(* Logix 5000 project; controller ExampleFile_V32 vendor 1 type 14 code 222 rev 32.11; software revision 32.00 *)

TASK MainTask (continuous, watchdog 500 ms) : MainProgram
TASK SafetyTask (periodic, rate 20 ms, priority 10, watchdog 20 ms, safety) : SafetyProgram

MODULES
   Local : vendor 1 type 14 code 222 (5069 0, rev 32.11)
END_MODULES

TYPE CommandString :   // Premixer command string based on CommandString.xlsx
STRUCT
   Cmd : STRING[10];
   Value : DINT[10];
END_STRUCT
END_TYPE

TYPE ISA88_PackML_Cmd :
STRUCT
   ClearFaults : BOOL;   // Program call to ClearFaults
   Clearing_ons : BOOL;   // Initialize to ClearFaults
   Hold_EM_Clear : TIMER;   // Holding time EM_Clear
   Resetting : BOOL;   // Program call to Resetting
   Resetting_ons : BOOL;   // Initialize Resetting
   Starting : BOOL;   // Program call to Starting
   Starting_ons : BOOL;   // Initialize Starting
   Stopping : BOOL;   // Program call to Stopping
   Stopping_ons : BOOL;   // Initialize Stopping
END_STRUCT
END_TYPE

TYPE ISA88_PackML_PackTags_Command :
STRUCT
   OpperationMode : ISA88_PackML_PackTags_Command_Opperation;   // Forces mode to obj model
   StateTransmittion : ISA88_State_UserInputs;
   Recept : DINT;   // currently not in use
END_STRUCT
END_TYPE

TYPE ISA88_PackML_PackTags_Command_Opperation :
STRUCT
   Automatic : BOOL;   // Forces mode to Automatic
   Maintenance : BOOL;   // Forces mode to Maintenance
   Manual : BOOL;   // Forces mode to Manual
   Cleaning : BOOL;   // Forces mode to Cleaning
   MES_Controlled : BOOL;   // Forces mode to CustomerDefined1
   CustomerDefined2 : BOOL;   // Forces mode to CustomerDefined2
END_STRUCT
END_TYPE

TYPE ISA88_PackML_PackTags_Status_Mode :   // Feedback which mode is active
STRUCT
   Automatic : BOOL;   // Current mode is Automatic
   Maintenance : BOOL;   // Current mode is Maintenance
   Manual : BOOL;   // Current mode is Manual
   Cleaning : BOOL;   // Current mode is Cleaning
   MES_Controlled : BOOL;   // Current mode is CustomerDefined1
   CustomerDefined2 : BOOL;   // Current mode is CustomerDefined2
END_STRUCT
END_TYPE

TYPE ISA88_PackML_SEQ :
STRUCT
   Clear : DINT;   // Clearing step number
   Resetting : DINT;   // Resetting step number
   Starting : DINT;   // Starting step number
   Stopping : DINT;   // Stopping step number
END_STRUCT
END_TYPE

TYPE ISA88_PackML_STS :
STRUCT
   ClearSeq_PC : BOOL;   // Clearing complete
   CompletingSeq_PC : BOOL;   // Completing complete
   ResettingSeq_PC : BOOL;   // Resetting complete
   StartingSeq_PC : BOOL;   // Starting complete
   StoppingSeq_PC : BOOL;   // Stopping complete
END_STRUCT
END_TYPE

TYPE ISA88_State_SC :
STRUCT
   Execute_to_Completing : BOOL;   // EquipmentModule requests to move from Execute to Completing
   Unholding_to_Execute : BOOL;   // EquipmentModule requests to move from Unholding to Execute
   Starting_to_Execute : BOOL;   // EquipmentModule requests to move from Starting to Execute
   Holding_to_Held : BOOL;   // EquipmentModule requests to move from Holding to Held
   Completing_to_Completed : BOOL;   // EquipmentModule requests to move from Completing to Completed
   Suspending_to_Suspended : BOOL;   // EquipmentModule requests to move from Suspending to Suspended
   Unsuspending_to_Execute : BOOL;   // EquipmentModule requests to move from Unsuspending to Execute
   Resetting_to_Idle : BOOL;   // EquipmentModule requests to move from Resetting to Idle
   Stopping_to_Stopped : BOOL;   // EquipmentModule requests to move from Stopping to Stopped
   Clearing_to_Stopped : BOOL;   // EquipmentModule requests to move from Clearing to Stopped
   Aborting_to_Aborted : BOOL;   // EquipmentModule requests to move from Aborting to Aborted
   Wrk_Module_Disabled : BOOL;   // Disables the module
   Wrk_Stop_trigger : BOOL;   // Forces the module to Stopped
   Wrk_Abort_trigger : BOOL;   // Forces the module to fault
   Sts_CurrentJob : STRING;   // Description of current job
   Wrk_Suspend : BOOL;   // Forces the module to suspend
   Wrk_Unsuspend : BOOL;   // Forces the module to Execute from Suspend
END_STRUCT
END_TYPE

TYPE ISA88_State_UserInputs :   // operations from the HMI
STRUCT
   Hold : BOOL;
   UnHold : BOOL;
   Start : BOOL;
   Suspend : BOOL;
   UnSuspend : BOOL;
   Reset : BOOL;
   Stop : BOOL;
   Abort : BOOL;
   Clear : BOOL;
END_STRUCT
END_TYPE

TYPE ISA88_State_UserOutputs :
STRUCT
   Held : BOOL;
   Unholding : BOOL;
   Holding : BOOL;
   Idle : BOOL;
   Starting : BOOL;
   Execute : BOOL;
   Completing : BOOL;
   Complete : BOOL;
   Resetting : BOOL;
   Unsuspending : BOOL;
   Suspended : BOOL;
   Suspending : BOOL;
   Stopped : BOOL;
   Stopping : BOOL;
   Clearing : BOOL;
   Aborted : BOOL;
   Aborting : BOOL;
END_STRUCT
END_TYPE

TYPE STRING16 :
STRUCT
   LEN : DINT;
   DATA : SINT[16];
END_STRUCT
END_TYPE

ADD_ON_INSTRUCTION ClearString   (* revision 1.0 *)
VAR_INPUT
   StartValue : DINT; {visible}
   final_value : DINT; {visible}
END_VAR
VAR_IN_OUT
   String : STRING[100]; {required}
END_VAR
VAR_INPUT
   cmd_Clear : BOOL; {visible}
END_VAR
VAR
   i : DINT; {access None}   // local index
END_VAR

ROUTINE Logic   (* structured text *)
   ////////////////////////////////////////////////////////////
   //   Copyright (c)
   //------------------------------------------------------------
   //   Routine: ClearString - Logic
   //   Author: WPI\tom.reit
   //   Created: 19-5-2022
   //------------------------------------------------------------
   //   Description:
   //
   //
   //   History:
   //
   ////////////////////////////////////////////////////////////
   if cmd_Clear then
   	for i := StartValue to final_value do
   		String[i]:='';
   	end_for;
   	cmd_Clear:=0;
   end_if;
END_ROUTINE
END_ADD_ON_INSTRUCTION

ADD_ON_INSTRUCTION Command_String   (* revision 1.0, vendor WPI, ExecutePrescan *)
// Mixer control based on Orklas command string.
// Revision note:
// First version
VAR_IN_OUT
   CommandString : STRING; {required}   // Input Command string
END_VAR
VAR_OUTPUT
   Cmd_Mixer : INT; {visible}   // bit 0 = stop mixer bit 1 = start mixer bit 2 = open mixer bit 3 = close mixer bit 4 = manual step bit 5 = discharge
   Cmd_Mixer_Speed_Fast : DINT; {visible}
   Cmd_Mixer_Time_Fast : DINT; {visible}
   Cmd_Mixer_Time_Slow : DINT; {visible}
   Cmd_Mixer_Time_Wait : DINT; {visible}
   Cmd_Mixer_Temperature : REAL; {visible}
   Cmd_Mixer_Time_Min : DINT; {visible}   // minimal mixing time
   Cmd_Mixer_Time_Max : DINT;   // max mixing time
   Sts_Time_RecievedCommand : LINT; {visible}
   Sts_Time_WriteCommand : LINT; {visible}
   Sts_MixingByTime : BOOL; {visible}
   Sts_MixingByTemperature : BOOL; {visible}
   Sts_SuccesfulRead : BOOL; {visible}   // String was succesful read and write according to CommandString
   ERR_InvalidCommand : BOOL; {visible}   // command didnt have end token
   ERR_TooManySegments : BOOL; {visible}   // Segment index reached higher than max value
   Cmd_Mixer_Speed_Slow : DINT; {visible}
END_VAR
VAR
   CommandString_Segment : STRING[10] := ([0] := 'MBD', [1] := 'MC', [2] := 'MSF', [3] := 'MTF');
   CommandString_Segment_Value : STRING[10] := ([0] := '1', [1] := '1', [2] := '80', [3] := '100');
   CommandStringSize : DINT := 26;
   count : INT := 82;
   i : INT;
   FoundPlace : DINT := 4;
   prev_i : DINT := 26;
   readString : BOOL;
   segment_Index : INT := 4;   // index num for array
   wrk_end_token : SINT := '#';   // end token will always be " # "
   wrk_split_token : SINT := ';';
   sts_CommandString : CommandString := (Cmd[0] := 'MBD', Cmd[1] := 'MC', Cmd[2] := 'MSF', Cmd[3] := 'MTF', Value[0] := 1, Value[1] := 1, Value[2] := 80, Value[3] := 100);
   wrk_String : STRING;   // temp string will be overwritten by each segment
   wrk_value_token_str : STRING := '_';
   wrk_Prev_CommandString : STRING;
END_VAR

ROUTINE Logic   (* structured text *)
// Mixer control based on Orklas command string.
   ////////////////////////////////////////////////////////////
   //   Copyright (c)  WPI
   //------------------------------------------------------------
   //   Routine: Command_String - Logic
   //   Author: WPI\engineer
   //   Created: 29-9-2021
   //------------------------------------------------------------
   //   Description:
   //           Mixer control based on Orklas command string.
   //
   //
   //   History:
   //
   ////////////////////////////////////////////////////////////
   #region "Check for new command"
   	if wrk_Prev_CommandString <> CommandString then
   		Sts_SuccesfulRead	:=0;
   		readString			:=1;
   		gsv(WallClockTime,,CurrentValue,Sts_Time_RecievedCommand);
   	end_if;
   #endregion
   #region "Read command string and apply logic"
   	if readString then
   	#region "Check if command is valid"
   		for i := 0 to 81 do
   			if CommandString.DATA[i] = wrk_end_token then
   				CommandStringSize		:=	i;	// set comamndstringSize
   				ERR_InvalidCommand		:=	0;	// valid string detected
   				exit;							// break for loop
   			end_if;
   			if i=81 AND CommandString.DATA[i] <> wrk_end_token then
   				ERR_InvalidCommand		:=	1; 	// no # was found in command string
   				readString				:=	0;	// break readstring
   			end_if;
   		end_for;
   				i						:=	0;	// set index back to 0
   	#endregion
   	#region Clear old Segments
   		for i := 0 to 9 do
   			Cmd_Mixer										:=0;
   			Cmd_Mixer_Speed_Fast							:=0;
   			Cmd_Mixer_Speed_Slow							:=0;
   			Cmd_Mixer_Temperature							:=0;
   			Cmd_Mixer_Time_Fast								:=0;
   			Cmd_Mixer_Time_Max								:=0;
   			Cmd_Mixer_Time_Min								:=0;
   			Cmd_Mixer_Time_Slow								:=0;
   			Cmd_Mixer_Time_Wait								:=0;
   			CommandString_Segment[i]						:='';
   			sts_CommandString.Cmd[i]						:='';
   			for count := 0 to 81 do
   				CommandString_Segment[i].DATA[count]		:=0;
   				sts_CommandString.Cmd[i].DATA[count]		:=0;
   				CommandString_Segment[i].LEN				:=0;
   				sts_CommandString.Cmd[i].LEN				:=0;
   				CommandString_Segment_Value[i].DATA[count]	:=0;
   				sts_CommandString.Cmd[i].DATA[count]		:=0;
   				CommandString_Segment_Value[i].LEN 			:=0;
   				sts_CommandString.Cmd[i].LEN 				:=0;
   			end_for;
   		end_for;
   		i:=0;
   	#endregion
   	#region ReadString
   		prev_i			:=	0;	// prepre for new string
   		segment_Index	:=	0;	// prepare for new string
   		for i := 0 to CommandStringSize do
   			wrk_String.DATA[i-prev_i]	:=	CommandString.DATA[i];
   			wrk_String.LEN				:=	i-prev_i;
   			if CommandString.DATA[i] = wrk_split_token  then
   				prev_i:=(i+1);
   				#region Prevent overflow array
   					if segment_Index>9 then
   						ERR_TooManySegments	:=1;
   						readString			:=0;
   						exit;
   					else
   						ERR_TooManySegments:=0;
   					end_if;
   				#endregion
   				CommandString_Segment[segment_Index]:=wrk_String;
   				segment_Index:=segment_Index+1;
   			end_if;
   		end_for;
   	#endregion
   	if NOT ERR_TooManySegments AND NOT ERR_InvalidCommand THEN
   		/* Clear wrk_string*/
   		wrk_String		:=	'';
   		wrk_String.LEN	:=	0;
   		#region read cmd value
   		FoundPlace:=0;
   		i:=0;
   			for i := 0 to segment_Index-1 do
   				find(CommandString_Segment[i],wrk_value_token_str,1,FoundPlace);
   				for count := FoundPlace to CommandString_Segment[i].LEN do
   					CommandString_Segment_Value[i].DATA[count-FoundPlace]:=CommandString_Segment[i].DATA[count];
   					CommandString_Segment_Value[i].LEN:=CommandString_Segment[i].LEN-FoundPlace;
   				end_for;
   			end_for;
   			i		:=	0;
   			count	:=	0;
   		#endregion
   		#region SubString
   			for i := 0 to segment_Index-1 do
   				find(CommandString_Segment[i],wrk_value_token_str,1,FoundPlace);
   				for count := FoundPlace-1 to 81 do
   					CommandString_Segment[i].DATA[count]:=0;
   				end_for;
   				CommandString_Segment[i].LEN:=FoundPlace-1;
   			end_for;
   		#endregion
   		#region Move values to sturcture
   			for i := 0 to segment_Index-1 do
   				sts_CommandString.Cmd[i]	:=	CommandString_Segment[i];
   				STOD(CommandString_Segment_Value[i],sts_CommandString.Value[i]);
   			end_for;
   		#endregion
   		#region "decode string"
   			for i := 0 to 9 do
   				if 		sts_CommandString.Cmd[i] 		= 	'MBD' 	then 	// Mixing by time / duration
   							Sts_MixingByTime:=1;
   							Sts_MixingByTemperature:=0;
   				elsif 	sts_CommandString.Cmd[i] 		= 	'MBT' 	then 	// Mixing by temperature
   							Sts_MixingByTime:=0;
   							Sts_MixingByTemperature:=1;
   				elsif 	sts_CommandString.Cmd[i] 		= 	'MC' 	then 	// Mixing Command
   					if		sts_CommandString.Value[i]	= 	0 		then	// Stop Mixer
   						Cmd_Mixer:=2#0000_0000_0000_0001;
   					elsif	sts_CommandString.Value[i]	= 	1 		then	// Start Mixer
   						Cmd_Mixer:=2#0000_0000_0000_0010;
   					elsif	sts_CommandString.Value[i]	= 	2 		then	// open Mixer
   						Cmd_Mixer:=2#0000_0000_0000_0100;
   					elsif	sts_CommandString.Value[i]	= 	3 		then	// close Mixer
   						Cmd_Mixer:=2#0000_0000_0000_1000;
   					elsif	sts_CommandString.Value[i]	= 	4 		then	// manual step active
   						Cmd_Mixer:=2#0000_0000_0001_0000;
   					elsif	sts_CommandString.Value[i]	= 	5 		then	// discharge mixer
   						Cmd_Mixer:=2#0000_0000_0010_0000;
   					end_if;
   				elsif 	sts_CommandString.Cmd[i] 		= 	'MSF' 	then 	// Mixer speed fast
   							Cmd_Mixer_Speed_Fast:=sts_CommandString.Value[i];
   				elsif 	sts_CommandString.Cmd[i] 		= 	'MSS' 	then 	// Mixer speed slow
   							Cmd_Mixer_Speed_Slow:=sts_CommandString.Value[i];
   				elsif 	sts_CommandString.Cmd[i] 		= 	'MTF' 	then 	// Mixing time fast
   							Cmd_Mixer_Time_Fast:=sts_CommandString.Value[i];
   				elsif 	sts_CommandString.Cmd[i] 		= 	'MTS' 	then 	// Mixing time slow
   							Cmd_Mixer_Time_Slow:=sts_CommandString.Value[i];
   				elsif 	sts_CommandString.Cmd[i] 		= 	'MTW' 	then 	// Waiting time
   							Cmd_Mixer_Time_Wait:=sts_CommandString.Value[i];
   				elsif 	sts_CommandString.Cmd[i] 		= 	'MOT' 	then 	// Optimal mixing temperature
   							Cmd_Mixer_Temperature:=sts_CommandString.Value[i];
   				elsif 	sts_CommandString.Cmd[i] 		= 	'MIT' 	then 	// Min mixing time
   							Cmd_Mixer_Time_Min:=sts_CommandString.Value[i];
   				elsif 	sts_CommandString.Cmd[i] 		= 	'MAT' 	then 	// Max mixing time
   							Cmd_Mixer_Time_Max:=sts_CommandString.Value[i];
   				end_if;
   			end_for;
   			Sts_SuccesfulRead:=1;
   			gsv(WallClockTime,,CurrentValue,Sts_Time_WriteCommand);
   		end_if;
   	#endregion
   	i:=0;
   	readString:=0;
   	wrk_Prev_CommandString:=CommandString;
   	end_if;
   #endregion
   
END_ROUTINE

ROUTINE Prescan   (* structured text *)
   ////////////////////////////////////////////////////////////
   //   Copyright (c)  WPI
   //------------------------------------------------------------
   //   Routine: Prescan
   //   Author: WPI\engineer
   //   Created: 29-9-2021
   //------------------------------------------------------------
   //   Description:
   //
   //
   //   History:
   //
   ////////////////////////////////////////////////////////////
   wrk_end_token		:=35; // 35 is # ascii
   wrk_split_token		:=59; // 35 is # ascii
   wrk_value_token_str	:='_';// _ is value token
   
   
END_ROUTINE
END_ADD_ON_INSTRUCTION

ADD_ON_INSTRUCTION CountUpAndDown   (* revision 1.0, vendor WPI *)
VAR_INPUT
   CountingSpeed : DINT; {visible}   // in miliseconds
END_VAR
VAR_OUTPUT
   Count : DINT; {visible}
END_VAR
VAR_INPUT
   MaxCount : DINT := 10; {visible}   // max value to count to
   Holding_Time : DINT := 2500; {visible}   // in milisec
END_VAR
VAR_OUTPUT
   Done : BOOL; {visible}
END_VAR
VAR
   Time_puls : TIMER := (PRE := 500); {access None}
   count_UP : BOOL := 1; {access None}
   holdingtime : TIMER[2]; {access None}
END_VAR

ROUTINE Logic   (* ladder *)
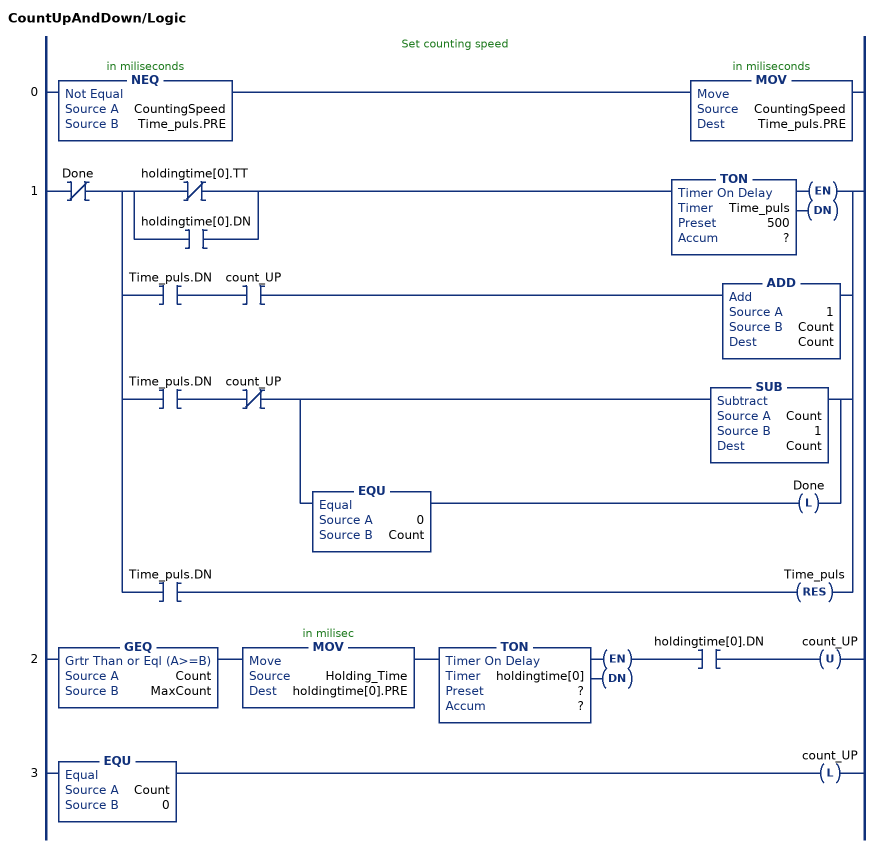
   // Set counting speed
   0: NEQ(CountingSpeed,Time_puls.PRE)MOV(CountingSpeed,Time_puls.PRE);
   1: XIO(Done)[[XIO(holdingtime[0].TT) ,XIC(holdingtime[0].DN) ] TON(Time_puls,?,?) ,XIC(Time_puls.DN) XIC(count_UP) ADD(1,Count,Count) ,XIC(Time_puls.DN) XIO(count_UP) [SUB(Count,1,Count) ,EQU(0,Count) OTL(Done) ] ,XIC(Time_puls.DN) RES(Time_puls) ];
   2: GEQ(Count,MaxCount)MOV(Holding_Time,holdingtime[0].PRE)TON(holdingtime[0],?,?)XIC(holdingtime[0].DN)OTU(count_UP);
   3: EQU(Count,0)OTL(count_UP);
END_ROUTINE
END_ADD_ON_INSTRUCTION

ADD_ON_INSTRUCTION CREATE_MERKER   (* revision 1.0 *)
VAR_INPUT
   INPUT : BOOL := 1; {required}
   RESET : BOOL; {required}
END_VAR
VAR_OUTPUT
   MERKER : BOOL; {access Read Only, visible}
END_VAR
VAR_INPUT
   I_NORMALY_OPEN : BOOL; {required}
END_VAR

ROUTINE Logic   (* ladder *)
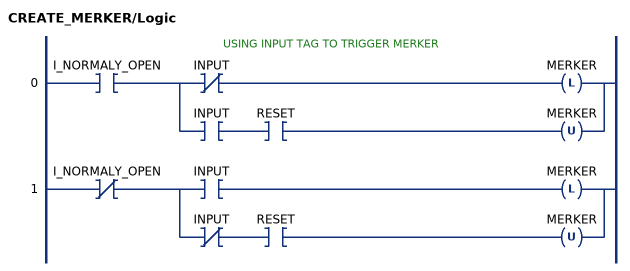
   // USING INPUT TAG TO TRIGGER MERKER
   0: XIC(I_NORMALY_OPEN)[XIO(INPUT) OTL(MERKER) ,XIC(INPUT) XIC(RESET) OTU(MERKER) ];
   1: XIO(I_NORMALY_OPEN)[XIC(INPUT) OTL(MERKER) ,XIO(INPUT) XIC(RESET) OTU(MERKER) ];
END_ROUTINE
END_ADD_ON_INSTRUCTION

ADD_ON_INSTRUCTION Dryrun_Sensor   (* revision 1.0, vendor WPI, ExecutePrescan *)
// Help:
// Geeft een alarm als de dryrun sensor 0 is en de pomp stuur waarde1 is.
VAR_INPUT
   I_DryrunSensor : BOOL; {required}
   I_PumpRunning : BOOL; {required}
END_VAR
VAR_OUTPUT
   Alarm : BOOL; {visible}   // Dryun is active
END_VAR
VAR_INPUT
   Reset : BOOL; {required}   // Reset the alarm if active
END_VAR
VAR
   DryrunTimer : TIMER := (PRE := 5000); {access None}
   ons : DINT; {access None}
END_VAR

ROUTINE Logic   (* ladder *)
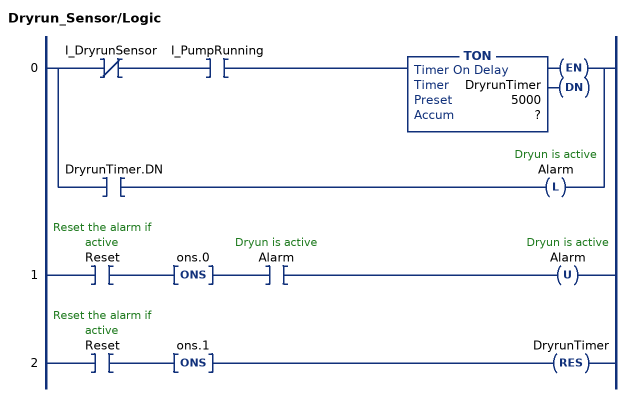
   0: [XIO(I_DryrunSensor) XIC(I_PumpRunning) TON(DryrunTimer,?,?) ,XIC(DryrunTimer.DN) OTL(Alarm) ];
   1: XIC(Reset)ONS(ons.0)XIC(Alarm)OTU(Alarm);
   2: XIC(Reset)ONS(ons.1)RES(DryrunTimer);
END_ROUTINE

ROUTINE Prescan   (* structured text *)
// sets timer
   DryrunTimer.PRE :=5000;		// set dryrun timer to 5 sec
END_ROUTINE
END_ADD_ON_INSTRUCTION

ADD_ON_INSTRUCTION FLIP_FLOP   (* revision 1.0 *)
VAR_INPUT
   input_time : DINT := 1500;
END_VAR
VAR_OUTPUT
   Q : BOOL; {access Read Only, visible}
   QB : BOOL; {access Read Only, visible}
END_VAR
VAR_INPUT
   INPUT_TIME_Q : DINT; {required}   // the time Q is going to be active
   INPUT_TIME_QB : DINT; {required}   // the time QB is going to be active
END_VAR
VAR
   FLIPFLOP_TIME : DINT; {access None}
   FLIPFLOP_timer1 : TIMER; {access None}
   FLIPFLOP_timer2 : TIMER := (PRE := 7500); {access None}
   FLIPFLOP_TIME1 : DINT; {access None}
   FLIPFLOP_TIME2 : DINT; {access None}
END_VAR

ROUTINE Logic   (* ladder *)
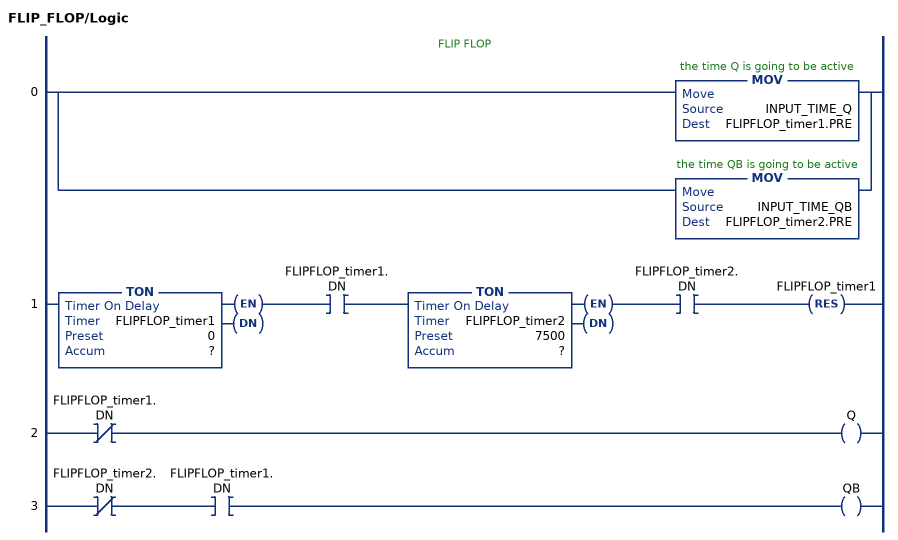
   // FLIP FLOP
   0: [MOV(INPUT_TIME_Q,FLIPFLOP_timer1.PRE) ,MOV(INPUT_TIME_QB,FLIPFLOP_timer2.PRE) ];
   1: TON(FLIPFLOP_timer1,?,?)XIC(FLIPFLOP_timer1.DN)TON(FLIPFLOP_timer2,?,?)XIC(FLIPFLOP_timer2.DN)RES(FLIPFLOP_timer1);
   2: XIO(FLIPFLOP_timer1.DN)OTE(Q);
   3: XIO(FLIPFLOP_timer2.DN)XIC(FLIPFLOP_timer1.DN)OTE(QB);
END_ROUTINE
END_ADD_ON_INSTRUCTION

ADD_ON_INSTRUCTION HMI_DIG_Sensor   (* revision 1.0, vendor WPI *)
// Help:
// 0 = NO
// 1 = NC
VAR_INPUT
   NC_or_NO_Mode : BOOL; {visible}   // 0 = NC 1 = NO
   Input : BOOL; {required}
   reset : BOOL; {required}
END_VAR
VAR_OUTPUT
   Alarm : BOOL; {access Read Only, visible}
END_VAR
VAR_INPUT
   Simulatie : BOOL; {visible}
   SimulatieValue : BOOL; {visible}
END_VAR
VAR
   C_M : CREATE_MERKER := (INPUT := 1); {access None}   // Create Merker
   NC_NO : BOOL; {access None}   // Normaly open or Normaly Closed 0= NC 1 = NO
   split_char : STRING; {access None}
   Found_location : DINT; {access None}
   Num_res : DINT; {access None}
   UpperTag : STRING16; {access None}
   LowerTag : STRING16; {access None}
END_VAR

ROUTINE Logic   (* ladder *)
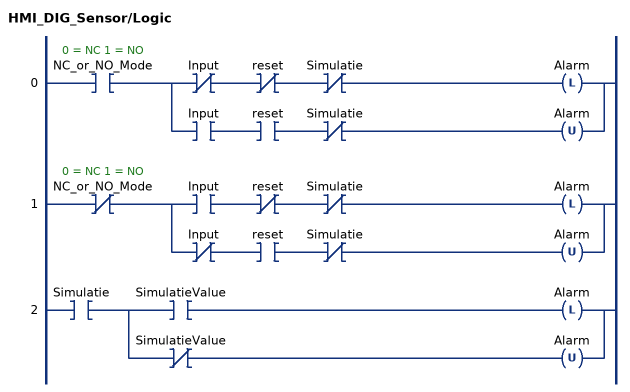
   0: XIC(NC_or_NO_Mode)[XIO(Input) XIO(reset) XIO(Simulatie) OTL(Alarm) ,XIC(Input) XIC(reset) XIO(Simulatie) OTU(Alarm) ];
   1: XIO(NC_or_NO_Mode)[XIC(Input) XIO(reset) XIO(Simulatie) OTL(Alarm) ,XIO(Input) XIC(reset) XIO(Simulatie) OTU(Alarm) ];
   2: XIC(Simulatie)[XIC(SimulatieValue) OTL(Alarm) ,XIO(SimulatieValue) OTU(Alarm) ];
END_ROUTINE
END_ADD_ON_INSTRUCTION

ADD_ON_INSTRUCTION IA_SENSOR   (* revision 2.0, vendor WPI *)
// Revision note:
// Tested by Tom Reit 25-2-2020
// Help:
// This addon instruction scales an analog input from a sensor.
// InRawMax, default: 16383 (20mA)
// InRawMin, default:  3277(4mA)
// InEUMax, max sensor value
// InEUmin, min sensor value
// RawSensorValue, this is the sensor analog input
// MODULE_ENABLE, this enables the module.
// SIMULATIE_ENABLE, if this is set to (TRUE/1) the scaling will be ignored and the OUTPUT will be the same as SIMULATIE_VALUE
VAR_INPUT
   InRawMax : REAL; {required}   // MAX analog value
   InRawMin : REAL; {required}   // MIN analog value
   InEUMax : REAL; {required}   // MAX scaled value
   InEUMin : REAL; {required}   // MIN scaled value
   RawSensorValue : REAL; {required}   // raw sensor value
   MODULE_ENABLE : BOOL; {required}   // TURNS ON THE MODULE
   SIMULATIE_ENABLE : BOOL; {required}   // Turns on the simulation and ignores the RawSensorValue
   SIMULATIE_VALUE : REAL; {required}   // Simulation value (make sure it is in the same range to achieve best preformance)
END_VAR
VAR_OUTPUT
   OUTPUT : REAL; {access Read Only, visible}   // Live Output value from the addon
END_VAR
VAR
   SCL_01 : SCALE; {access None}
   SEL_01 : SELECT; {access None}
   ScaledSensorValue : REAL;   // scaled value
   __l71F380F08DE35724 : REAL; {access None}
   __lD3D84D0C4261A5C0 : REAL; {access None}
   __l18DEFF66D7D8D2CC : REAL; {access None}
   __l546263A5BCF0B27A : REAL; {access None}
   __lCCD375A3821135C8 : BOOL; {access None}
   __l32A3E1D26247E00E : REAL; {access None}
   __l255F8420B0BBFEF3 : BOOL; {access None}
   __l60D01122123B8153 : REAL; {access None}
   __lAE68D78140BEC49D : REAL; {access None}
   __foutF9DF9AFBB9497D4A : BOOL[32]; {access None}
END_VAR

ROUTINE Logic   (* function block diagram *)
   SHEET 1
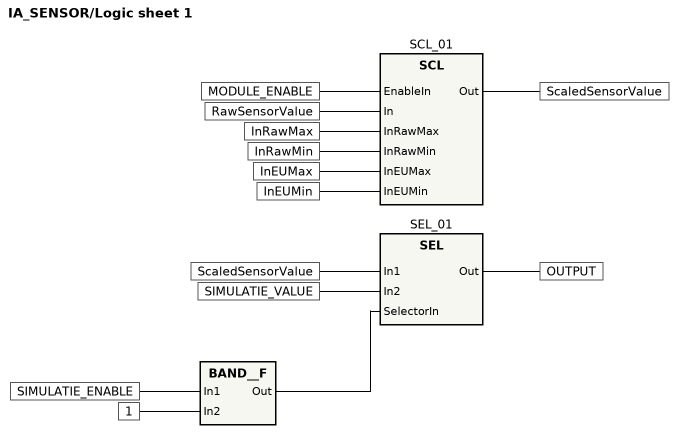
   BAND__F_1 : BAND__F(In1 := SIMULATIE_ENABLE, In2 := 1);
   SCL_01 : SCL(EnableIn := MODULE_ENABLE, In := RawSensorValue, InRawMax := InRawMax, InRawMin := InRawMin, InEUMax := InEUMax, InEUMin := InEUMin);
   SEL_01 : SEL(In1 := ScaledSensorValue, In2 := SIMULATIE_VALUE, SelectorIn := BAND__F_1.Out);
   ScaledSensorValue := SCL_01.Out;
   OUTPUT := SEL_01.Out;
END_ROUTINE
END_ADD_ON_INSTRUCTION

ADD_ON_INSTRUCTION ProductBuffer_V2   (* revision 1.0 *)
// including user defined overflow
VAR_IN_OUT
   Buffer : REAL[100]; {required}
END_VAR
VAR_OUTPUT
   ProductAmount : DINT; {access Read Only, visible}   // products in buffer
   ER_Overflow : DINT; {access Read Only, visible}   // array over flow occoured
END_VAR
VAR_INPUT
   Reset : BOOL; {visible}
   bufferEnabled : BOOL; {visible}
   ProductDetect : BOOL; {required}
   HMI_SimulateProductDetect : BOOL; {visible}
END_VAR
VAR_OUTPUT
   ProductReachedObject : BOOL; {access Read Only, visible}
END_VAR
VAR_INPUT
   ActualPosition : REAL; {required}   // most likely the conveyor position
   Distance_to_Object : REAL; {required}   // distance from detection to object
END_VAR
VAR_OUTPUT
   RemainingDistance : REAL; {access Read Only, visible}
END_VAR
VAR_INPUT
   WrapAroundPosition : REAL; {required}   // this is the point where the value of actualPosition overflows / wrapsaround
END_VAR
VAR
   MAX_ARRAY_SIZE : DINT; {access None}
   RE_productDetect : FBD_ONESHOT; {access None}
   i : DINT; {access None}   // index num
   wrk_calculated_Position : REAL; {access None}
   detect_A : REAL; {access None}
   detect_B : REAL; {access None}
   wrk_buffershift : DINT; {access None}
END_VAR

ROUTINE Logic   (* structured text *)
// including user defined overflow
   ////////////////////////////////////////////////////////////
   //   Copyright (c)
   //------------------------------------------------------------
   //   Routine: ProductBuffer_V2 - Logic
   //   Author: WPI\tom.reit
   //   Created: 22-4-2022
   //------------------------------------------------------------
   //   Description:
   //           including user defined overflow
   //
   //
   //   History:
   //
   ////////////////////////////////////////////////////////////
   if s:fs then size(Buffer[0],0,MAX_ARRAY_SIZE); end_if;					// get buffersize
   
   /* Function list */
   OSRI(RE_productDetect);
   
   #region Prevent overflow
   	if i=0 					 then		i:=1; 									end_if;// prevents underflow
   	if (i>=MAX_ARRAY_SIZE-1) then		i:=MAX_ARRAY_SIZE-1; ER_Overflow:=1;	end_if;// prevents overflow
   	ProductAmount:=i-1;																   // indicator how many products are in buffer.
   #endregion
   #region Clear buffer
   	if Reset then
   		ER_Overflow:=0;											// reset error from overflow
   		for i:= 0 to MAX_ARRAY_SIZE-1 do
   			Buffer[i]:=WrapAroundPosition+1;					// set buffer element to wraparound +1 a position that can never be reached, because of wraparound.
   		end_for;
   		i:=0;
   	end_if;
   #endregion
   #region Enable Buffer
   	if bufferEnabled then
   		RE_productDetect.InputBit := ProductDetect OR HMI_SimulateProductDetect;	// on the rising edge product will be added to buffer
   	else
   		ProductReachedObject:=0;
   		RE_productDetect.InputBit:=0;
   		RE_productDetect.OutputBit:=0;
   		//Reset:=1;
   	end_if;
   #endregion
   #region add product to buffer
   	if RE_productDetect.OutputBit then												// Product count and add to buffer
   		wrk_calculated_Position:=0;													// clear previous value
   		wrk_calculated_Position:=ActualPosition+Distance_to_Object;					// calculate end point.
   
   		/* check if value is valid within wraparound position. if not subtract the wraparound */
   		if wrk_calculated_Position >= WrapAroundPosition then
   			Buffer[i]:= (ActualPosition+Distance_to_Object)-WrapAroundPosition;		// add item to (buffer + distance) - wraparound
   		else
   			Buffer[i]:= (ActualPosition+Distance_to_Object);						// add item to buffer + distance.
   		end_if;
   		i:=i+1;																		// set index to next item in buffer.
   	end_if;
   #endregion
   #region Product reached object
   	/*
   		because we're dealing with a wraparound
   		we have to worry about buffer element was ouside wraparound, so got wrapped to lower position.
   		but the actual position did not wraparound yet.
   
   		so we cant just say if actualposition >= buffer[i]
   
   		to resolve this were using 2 points A & B.
   		A = ActualPosition
   		B = ActualPosition - 1
   
   		if A>=Buffer[1] && B < Buffer[1] product reached object. this means we only detect in forwards direction.
   	*/
   	detect_A:=ActualPosition;
   	detect_B:=ActualPosition-1;
   	if detect_A >= Buffer[1] AND Buffer[1] > detect_B then
   		if i <> 1 then
   			for wrk_buffershift := 0 to MAX_ARRAY_SIZE-2 do
   				Buffer[wrk_buffershift]:=Buffer[wrk_buffershift+1];
   			end_for;
   
   			i:=i-1;
   		else
   			i:=1;// only 1 item in buffer, so dont have to loop back
   		end_if;
   		ProductReachedObject:=1; // set to true.
   	end_if;
   #endregion
   #region HMI visuals
   	if Buffer[1] <> Buffer[2] then							// only check first element
   		RemainingDistance:=Buffer[1]-ActualPosition;		// update ramaing distance constantly
   	else
   		RemainingDistance:=0;								// if buffer is empty dont update remaining distance.
   	end_if;
   #endregion
END_ROUTINE
END_ADD_ON_INSTRUCTION

ADD_ON_INSTRUCTION Servo_Object   (* revision 1.2 *)
// Revision note:
// Added motion intrustions reset command, once reset is active set all flags back to 0. so no previous state is in memory. Also unlatch all input signals if they were previous active while error occoured.
VAR_IN_OUT
   Axis_Object : AXIS_CIP_DRIVE; {required}   // Axis to control / monitor
   Module : MODULE; {required}   // Servo Drive
END_VAR
VAR_OUTPUT
   Sts_Faulted : BOOL; {access Read Only, visible}   // Axis faulted, check faultlist for detailed information.
   Sts_Enabled : BOOL; {access Read Only, visible}   // Drive is enabled(MSO) and "Running"on drive display
   Sts_Disabled : BOOL; {access Read Only, visible}   // Drive is disabeld(MSF) and "Stopped" on drive display
   Sts_StandStill : BOOL; {access Read Only, visible}   // Axis is not in motion
END_VAR
VAR_IN_OUT
   Sts_FaultMessage : STRING; {required}   // Contains data about error and what coased it
END_VAR
VAR_INPUT
   Inp_Enable : BOOL; {visible}   // Set to true to enable the drive, once completed or faulted signal will be set low as feedback
   Inp_Reset : BOOL; {visible}   // User reset, most likely EM_Clear
   Inp_Disable : BOOL; {visible}   // Set to true to disable the drive, once completed or faulted signal will be set low as feedback
   Inp_Stop : BOOL; {visible}   // Stop current motion, if retreive lost postions is set to true, axis will move back to its stopping position)
   Cnf_DecelRate : REAL; {visible}   // based on user units per sec ²
   Cnf_DecelJerk : REAL; {visible}   // % of time
   Cnf_RetrieveStoppingPositions : BOOL; {visible}   // If set to true the servo will start its stopping sequence but after is done it will move back to the position where the stopping command was given. for example if the stopping motion coased 15 user units the axis will move back 15 units.
   Cnf_Retrieve_Accel : REAL; {visible}   // in user units per sec ² (accel and decel are the same for retrieve position)
   Cnf_Retrieve_Speed : REAL; {visible}   // Retrieve_Speed in user units per sec
END_VAR
VAR_IN_OUT
   PackML : ISA88_PackML; {required}
END_VAR
VAR
   SEQ_Enable : DINT; {access None}   // statemodel for enabling drive
   Error : BOOL; {access None}   // local error ocoured, check fault list
   TRUE : BOOL := 1; {access None}   // always 1 ( true)
   FALSE : BOOL; {access None}   // always 0( false)
   reset_ons : FBD_ONESHOT; {access None}   // falling edge function for reset
   MAFR_Axis : MOTION_INSTRUCTION; {access None}   // reset axis
   MSO_Axis : MOTION_INSTRUCTION; {access None}   // local MSO to turn on servo
   MSF_Axis : MOTION_INSTRUCTION; {access None}   // local turn off servo
   DriveStatus : DINT; {access None}
   Wrk_InhibitModule : DINT; {access None}   // Local mem to set object into certain mode
   Wrk_InhibitAxis : DINT; {access None}   // local mem to set axis in centain mode
   Wrk_ModuleFaultCode : DINT; {access None}   // local module fault code to generate FaultMessage
   Wrk_AxisFaultBits : DINT; {access None}   // local Axis fault code to generate FaultMessage
   Wrk_MotionFaultBits : DINT; {access None}   // local Axis fault code to generate FaultMessage
   S_ModuleFaultCode : STRING; {access None}   // String conversion
   S_AxisFaultBits : STRING := '$0D$0A'; {access None}   // Conversion
   S_MotionFaultBits : STRING; {access None}   // Conversion
   i : DINT; {access None}   // local index num
   temp_num : DINT; {access None}   // temporary number only used for calculations as step inbetween because studio 5000 is idiot software
   Wrk_FaultMessage : STRING; {access None}   // building string
   SEQ_Stopping : DINT; {access None}   // statemodel for stopping motion
   wrk_CurrentPosition : REAL; {access None}   // last position before stopping
   MAS_Axis : MOTION_INSTRUCTION; {access None}   // Stopping motion instruction
   wrk_Max_DecelRate : REAL; {access None}   // based on motion settings
   MAM_Axis : MOTION_INSTRUCTION; {access None}   // Retrieve postion motion instruction
   wrk_MaximumSpeed : REAL; {access None}   // local max speed
   Wrk_CIPAxisFault : LINT; {access None}   // local copy of CIPAxisFaults
   S_CIPAxisFault : STRING; {access None}   // Local string to add all CIP axis faults to
   Alarm_Texts : STRING[100] := ([0] := 'MotorOvercurrentFault$0D$0A', [1] := 'MotorCommutationFault$0D$0A', [2] := 'MotorOverspeedFLFault', [3] := 'MotorOverspeedULFault', [4] := 'MotorOvertemperatureFLFault', [5] := 'MotorOvertemperatureULFault', [6] := 'MotorThermalOverloadFLFault', [7] := 'MotorThermalOverloadULFault', [8] := 'MotorPhaseLossFault', [9] := 'InverterOvercurrentFault', [10] := 'InverterOvertemperatureFLFault', [11] := 'InverterOvertemperatureULFault', [12] := 'InverterThermalOverloadFLFault', [13] := 'InverterThermalOverloadULFault', [14] := 'ConverterOvercurrentFault', [15] := 'ConverterGroundCurrentFLFault', [16] := 'ConverterGroundCurrentULFault', [17] := 'ConverterOvertemperatureFLFault', [18] := 'ConverterOvertemperatureULFault', [19] := 'ConverterThermalOverloadFLFault', [20] := 'ConverterThermalOverloadULFault', [21] := 'ConverterACPowerLossFault', [22] := 'ConverterACSinglePhaseLossFault', [23] := 'ConverterACPhaseShortFault', [24] := 'ConverterPreChargeFault', [25] := 'BusRegulatorOvertemperatureFLFault', [26] := 'BusRegulatorOvertemperatureULFault', [27] := 'BusRegulatorThermalOverloadFLFault', [28] := 'BusRegulatorThermalOverloadULFault', [29] := 'BusRegulatorFault', [30] := 'BusModuleFault', [31] := 'BusUndervoltageFLFault', [32] := 'BusUndervoltageULFault', [33] := 'BusOvervoltageFLFault', [34] := 'BusOvervoltageULFault', [35] := 'BusPowerLossFault', [36] := 'BusPowerBlownFuseFault', [37] := 'BusPowerLeakageFault', [38] := 'BusPowerSharingFault', [39] := 'FeedbackSignalNoiseFLFault', [40] := 'FeedbackSignalNoiseULFault', [41] := 'FeedbackSignalLossFLFault', [42] := 'FeedbackSignalLossULFault', [43] := 'FeedbackDataLossFLFault', [44] := 'FeedbackDataLossULFault', [45] := 'FeedbackDeviceFault', [46] := 'SensorFault', [47] := 'BrakeSlipFault', [48] := 'HardwareOvertravelPositiveFault', [49] := 'HardwareOvertravelNegativeFault', [50] := 'ExcessivePositionErrorFault', [51] := 'ExcessiveVelocityErrorFault', [52] := 'OvertorqueLimitFault', [53] := 'UndertorqueLimitFault', [54] := 'ExcessiveBusVoltageErrorFault', [55] := 'AmbientTemperatureRiseFault', [56] := 'IllegalControlModeFault', [57] := 'EnableInputDeactivatedFault', [58] := 'ControllerInitiatedFault', [59] := 'ExternalInputFault',
        [60] := 'Undefined Fault', [61] := 'Undefined Fault', [62] := 'Undefined Fault', [63] := 'spare'); {access None}   // Placeholder, just used to COP out of.
   Wrk_ModuleFaultBits : DINT; {access None}   // axis group module faults
   Wrk_AxisState : DINT; {access None}   // current axis state
   S_FaultCode_Base : STRING := 'Current Fault:'; {access None}   // contains begin of fault message
END_VAR

ROUTINE Logic   (* structured text *)
   ////////////////////////////////////////////////////////////
   //   Copyright (c)
   //------------------------------------------------------------
   //   Routine: Servo_Object - Logic
   //   Author: WPI\tom.reit
   //   Created: 6-5-2022
   //------------------------------------------------------------
   //   Description:
   //
   //
   //   History:
   //
   ////////////////////////////////////////////////////////////
   #region Macros
   	TRUE	:=1;
   	FALSE	:=0;
   #endregion
   #region Reset axis
   	OSFI(reset_ons);													// onshot (fallingedge) reset object
   	reset_ons.InputBit:=Inp_Reset;										// input reset signal
   	if reset_ons.OutputBit then MSO_Axis.FLAGS:=0; end_if;				// set MSO flags to 0.
   	if reset_ons.OutputBit then MSF_Axis.FLAGS:=0; end_if;				// set MSF flags to 0.
   	if reset_ons.OutputBit then MAM_Axis.FLAGS:=0; end_if;				// set MAM flags to 0.
   	if reset_ons.OutputBit then MAS_Axis.FLAGS:=0; end_if;				// set MAS flags to 0.
   
   	if reset_ons.OutputBit then SEQ_Enable:=0; end_if;					// set SEQ_Enable to 0.
   	if reset_ons.OutputBit then SEQ_Stopping:=0; end_if;				// set SEQ_Stopping to 0.
   
   	if Inp_Enable AND reset_ons.OutputBit AND Sts_Faulted 	then Inp_Enable	:=	FALSE; end_if;
   	if Inp_Disable AND reset_ons.OutputBit AND Sts_Faulted	then Inp_Disable:=	FALSE; end_if;
   	if Inp_Stop AND reset_ons.OutputBit AND Sts_Faulted		then Inp_Stop	:=	FALSE; end_if;
   
   	if reset_ons.OutputBit and Error then Error:=FALSE; end_if;			// if Error is active, set error to false.
   	if reset_ons.OutputBit then MAFR(Axis_Object,MAFR_Axis); end_if;	// Reset axis on output from reset signal.
   	if MAFR_Axis.ER AND MAFR_Axis.EN then Error:=TRUE; end_if;			// if while resetting axis fault occours, set Error back to true.
   #endregion
   #region Fault handler
   	//if Wrk_AxisState 					=8		then Error:=TRUE; end_if;	// tijdelijk uit
   	//if Wrk_AxisState 					=5		then Error:=TRUE; end_if;  // tijdelijk uit
   	if Axis_Object.MotionAlarmStatus	<>0 	then Error:=TRUE; end_if;
   	if Axis_Object.AxisFault			<>0 	then Error:=TRUE; end_if;
   	if Axis_Object.MotionFaultStatus	<>0		then Error:=TRUE; end_if;
   	if MSO_Axis.ER AND MSO_Axis.EN				THEN Error:=TRUE; end_if;
   	if MSF_Axis.ER AND MSF_Axis.EN				THEN Error:=TRUE; end_if;
   	if MAS_Axis.ER AND MAS_Axis.EN				THEN Error:=TRUE; end_if;
   	if MAM_Axis.ER AND MAM_Axis.EN				THEN Error:=TRUE; end_if;
   
   	Sts_Faulted:=Error;
   #endregion
   #region Drive Enable / Disable
   	if Inp_Enable 	AND SEQ_Enable=0 then SEQ_Enable:=10; end_if;
   	if Inp_Disable 	AND SEQ_Enable=0 then SEQ_Enable:=110; end_if;
   	case SEQ_Enable of
   		/*
   		state transmittions
   		 10 -> 40 	= Enable
   		110 -> 140 	= Disable
   		*/
   		0: /* waiting for command */
   			Sts_Enabled		:=		Axis_Object.DriveEnableStatus;
   			Sts_Disabled	:= NOT 	Axis_Object.DriveEnableStatus;
   		#region Enable drive
   		10: /* Recieve command from user, start enabling drive */
   			if 		Axis_Object.DriveEnableStatus then SEQ_Enable:=0; Sts_Enabled:=FALSE; 	end_if;// drive was already enabled.
   			if 	NOT Axis_Object.DriveEnableStatus then SEQ_Enable:=20; 	end_if;// drive was not enabled start enabling.
   
   		20: /* Check for servo faults, if there are any */
   			if 		Error then SEQ_Enable	:=999; 	end_if;
   			if NOT 	Error then SEQ_Enable	:=30; 	end_if;
   		30:	/* Enable servo */
   			MSO(Axis_Object,MSO_Axis);
   			SEQ_Enable:=35;
   		35: /* wait for feedback from MSO */
   			if MSO_Axis.EN AND MSO_Axis.DN then SEQ_Enable:=40; 	end_if;
   			if MSO_Axis.EN AND MSO_Axis.ER then SEQ_Enable:=999; 	end_if;
   		40:	/* Servo is enabled and ready to recieve commands */
   			if NOT 	Axis_Object.PowerStructureEnabledStatus then SEQ_Enable:=999; 	end_if;
   			if 		Axis_Object.PowerStructureEnabledStatus then
   				Inp_Enable:=FALSE;		// feedback to user, execution was done.
   				SEQ_Enable:=0;
   			end_if;
   		#endregion
   		#region Disable drive
   		110: /* Recieve command from user, start Disabling drive */
   			if 		Axis_Object.DriveEnableStatus then SEQ_Enable:=120; end_if;	// drive was not Disabled start disabling
   			if 	NOT Axis_Object.DriveEnableStatus then SEQ_Enable:=0; Inp_Disable:=FALSE; 	end_if;	// drive was already disabled.
   
   		120: /* Check for servo faults, if there are any */
   			if 		Error then SEQ_Enable	:=999; 	end_if;
   			if NOT 	Error then SEQ_Enable	:=130; 	end_if;
   		130:	/* Disable servo */
   			MSF(Axis_Object,MSF_Axis);
   			SEQ_Enable:=135;
   		135: /* wait for feedback from MSF */
   			if MSF_Axis.EN AND MSF_Axis.DN then SEQ_Enable:=140; 	end_if;
   			if MSF_Axis.EN AND MSF_Axis.ER then SEQ_Enable:=999; 	end_if;
   		140:	/* Servo is Disabeld and ready to recieve commands */
   			if  	Axis_Object.PowerStructureEnabledStatus then SEQ_Enable:=999; 	end_if;
   			if 	NOT	Axis_Object.PowerStructureEnabledStatus then
   				Inp_Disable:=FALSE;		// feedback to user, execution was done.
   				SEQ_Enable:=0;
   			end_if;
   		#endregion
   		999: /* Error state */
   			Inp_Enable:=FALSE;		// feedback to user, execution was done.
   			if reset_ons.OutputBit then SEQ_Enable:=0; end_if; // on reset set state back to 0.
   		else
   			SEQ_Enable:=0;// undefined state, goes to 0
   	end_case;
   #endregion
   #region (Un)Inhibit drive / (Un)Inhibit motion axis
   	/*
   		DriveStatus = 16#1000	// Faulted
   		DriveStatus = 16#4000	// running
   		DriveStatus = 16#6000	// inhibit
   	*/
   	GSV(Module,Module,EntryStatus,DriveStatus);					// Get entry status of module
   	if PackML.Disable_Module then
   		Wrk_InhibitModule	:=4; 	SSV(Module,Module,Mode,Wrk_InhibitModule);			// inhibbit module
   		Wrk_InhibitAxis		:=1; 	SSV(Axis,Axis_Object,InhibitAxis,Wrk_InhibitAxis); 	// inhibbit Axis
   	else
   		if DriveStatus = 16#6000 then
   			Wrk_InhibitModule	:=0; 	SSV(Module,Module,Mode,Wrk_InhibitModule);			// inhibbit module
   			Wrk_InhibitAxis		:=0; 	SSV(Axis,Axis_Object,InhibitAxis,Wrk_InhibitAxis); 	// inhibbit Axis
   		end_if;
   	end_if;
   #endregion
   #region Fault String
   
   	GSV(Module,Module,FaultCode,Wrk_ModuleFaultCode);
   	GSV(Axis,Axis_Object,AxisState,Wrk_AxisState);
   	GSV(Axis,Axis_Object,ModuleFaultBits,Wrk_ModuleFaultBits);
   	GSV(Axis,Axis_Object,AxisFaultBits,Wrk_AxisFaultBits);
   	GSV(Axis,Axis_Object,MotionFaultBits,Wrk_MotionFaultBits);
   	Wrk_CIPAxisFault:=Axis_Object.CIPAxisFaults;
   	/* Convert dints to String */
   	#region Clear strings using for loop to avoid using move etc, old plcs / older software versions 30 and below can't handle these operations, loser software verions
   		for i := 0 to 81 do
   			S_ModuleFaultCode.DATA[i]	:=	0;	// 0 DEC = '$00' ASCII
   			S_AxisFaultBits.DATA[i]		:=	0;	// 0 DEC = '$00' ASCII
   			S_MotionFaultBits.DATA[i]	:=	0;	// 0 DEC = '$00' ASCII
   			S_CIPAxisFault.DATA[i]		:=	0;	// 0 DEC = '$00' ASCII
   			Wrk_FaultMessage.DATA[i]	:=	0;	// 0 DEC = '$00' ASCII
   		end_for;
   		i:=0;									// set index to 0
   		S_CIPAxisFault.LEN		:=i;			// set String length to 0
   		Wrk_FaultMessage.LEN	:=i;			// set String length to 0
   		S_ModuleFaultCode.LEN	:=i;			// set String length to 0
   		S_AxisFaultBits.LEN		:=i;			// set String length to 0
   		S_MotionFaultBits.LEN	:=i;			// set String length to 0
   	#endregion
   	DTOS(Wrk_ModuleFaultCode,S_ModuleFaultCode);
   	DTOS(Wrk_AxisFaultBits,S_AxisFaultBits);
   	DTOS(Wrk_MotionFaultBits,S_MotionFaultBits);
   	#region build string
   		if 		Axis_Object.MotorOvercurrentFault 				then temp_num:=S_CIPAxisFault.LEN+1; INSERT(Alarm_Texts[0],S_CIPAxisFault,temp_num,S_CIPAxisFault); // 		Axis_Object.MotorOvercurrentFault
   		elsif  	Axis_Object.MotorCommutationFault 				then temp_num:=S_CIPAxisFault.LEN+1; INSERT(Alarm_Texts[1],S_CIPAxisFault,temp_num,S_CIPAxisFault); // 		Axis_Object.MotorCommutationFault
   		elsif  	Axis_Object.MotorOverspeedFLFault 				then temp_num:=S_CIPAxisFault.LEN+1; INSERT(Alarm_Texts[2],S_CIPAxisFault,temp_num,S_CIPAxisFault); // 		Axis_Object.MotorOverspeedFLFault
   		elsif  	Axis_Object.MotorOverspeedULFault 				then temp_num:=S_CIPAxisFault.LEN+1; INSERT(Alarm_Texts[3],S_CIPAxisFault,temp_num,S_CIPAxisFault); // 		Axis_Object.MotorOverspeedULFault
   		elsif  	Axis_Object.MotorOvertemperatureFLFault 		then temp_num:=S_CIPAxisFault.LEN+1; INSERT(Alarm_Texts[4],S_CIPAxisFault,temp_num,S_CIPAxisFault); // 		Axis_Object.MotorOvertemperatureFLFault
   		elsif  	Axis_Object.MotorOvertemperatureULFault 		then temp_num:=S_CIPAxisFault.LEN+1; INSERT(Alarm_Texts[5],S_CIPAxisFault,temp_num,S_CIPAxisFault); // 		Axis_Object.MotorOvertemperatureULFault
   		elsif  	Axis_Object.MotorThermalOverloadFLFault 		then temp_num:=S_CIPAxisFault.LEN+1; INSERT(Alarm_Texts[6],S_CIPAxisFault,temp_num,S_CIPAxisFault); // 		Axis_Object.MotorThermalOverloadFLFault
   		elsif  	Axis_Object.MotorThermalOverloadULFault 		then temp_num:=S_CIPAxisFault.LEN+1; INSERT(Alarm_Texts[7],S_CIPAxisFault,temp_num,S_CIPAxisFault); // 		Axis_Object.MotorThermalOverloadULFault
   		elsif  	Axis_Object.MotorPhaseLossFault 				then temp_num:=S_CIPAxisFault.LEN+1; INSERT(Alarm_Texts[8],S_CIPAxisFault,temp_num,S_CIPAxisFault); // 		Axis_Object.MotorPhaseLossFault
   		elsif  	Axis_Object.InverterOvercurrentFault 			then temp_num:=S_CIPAxisFault.LEN+1; INSERT(Alarm_Texts[9],S_CIPAxisFault,temp_num,S_CIPAxisFault); // 		Axis_Object.InverterOvercurrentFault
   		elsif  	Axis_Object.InverterOvertemperatureFLFault 		then temp_num:=S_CIPAxisFault.LEN+1; INSERT(Alarm_Texts[10],S_CIPAxisFault,temp_num,S_CIPAxisFault); // 	Axis_Object.InverterOvertemperatureFLFault
   		elsif  	Axis_Object.InverterOvertemperatureULFault 		then temp_num:=S_CIPAxisFault.LEN+1; INSERT(Alarm_Texts[11],S_CIPAxisFault,temp_num,S_CIPAxisFault); // 	Axis_Object.InverterOvertemperatureULFault
   		elsif  	Axis_Object.InverterThermalOverloadFLFault 		then temp_num:=S_CIPAxisFault.LEN+1; INSERT(Alarm_Texts[12],S_CIPAxisFault,temp_num,S_CIPAxisFault); // 	Axis_Object.InverterThermalOverloadFLFault
   		elsif  	Axis_Object.InverterThermalOverloadULFault 		then temp_num:=S_CIPAxisFault.LEN+1; INSERT(Alarm_Texts[13],S_CIPAxisFault,temp_num,S_CIPAxisFault); // 	Axis_Object.InverterThermalOverloadULFault
   		elsif  	Axis_Object.ConverterOvercurrentFault 			then temp_num:=S_CIPAxisFault.LEN+1; INSERT(Alarm_Texts[14],S_CIPAxisFault,temp_num,S_CIPAxisFault); // 	Axis_Object.ConverterOvercurrentFault
   		elsif  	Axis_Object.ConverterGroundCurrentFLFault 		then temp_num:=S_CIPAxisFault.LEN+1; INSERT(Alarm_Texts[15],S_CIPAxisFault,temp_num,S_CIPAxisFault); // 	Axis_Object.ConverterGroundCurrentFLFault
   		elsif  	Axis_Object.ConverterGroundCurrentULFault 		then temp_num:=S_CIPAxisFault.LEN+1; INSERT(Alarm_Texts[16],S_CIPAxisFault,temp_num,S_CIPAxisFault); // 	Axis_Object.ConverterGroundCurrentULFault
   		elsif  	Axis_Object.ConverterOvertemperatureFLFault 	then temp_num:=S_CIPAxisFault.LEN+1; INSERT(Alarm_Texts[17],S_CIPAxisFault,temp_num,S_CIPAxisFault); // 	Axis_Object.ConverterOvertemperatureFLFault
   		elsif  	Axis_Object.ConverterOvertemperatureULFault 	then temp_num:=S_CIPAxisFault.LEN+1; INSERT(Alarm_Texts[18],S_CIPAxisFault,temp_num,S_CIPAxisFault); // 	Axis_Object.ConverterOvertemperatureULFault
   		elsif  	Axis_Object.ConverterThermalOverloadFLFault 	then temp_num:=S_CIPAxisFault.LEN+1; INSERT(Alarm_Texts[19],S_CIPAxisFault,temp_num,S_CIPAxisFault); //	 	Axis_Object.ConverterThermalOverloadFLFault
   		elsif  	Axis_Object.ConverterThermalOverloadULFault 	then temp_num:=S_CIPAxisFault.LEN+1; INSERT(Alarm_Texts[20],S_CIPAxisFault,temp_num,S_CIPAxisFault); // 	Axis_Object.ConverterThermalOverloadULFault
   		elsif  	Axis_Object.ConverterACPowerLossFault 			then temp_num:=S_CIPAxisFault.LEN+1; INSERT(Alarm_Texts[21],S_CIPAxisFault,temp_num,S_CIPAxisFault); // 	Axis_Object.ConverterACPowerLossFault
   		elsif  	Axis_Object.ConverterACSinglePhaseLossFault 	then temp_num:=S_CIPAxisFault.LEN+1; INSERT(Alarm_Texts[22],S_CIPAxisFault,temp_num,S_CIPAxisFault); // 	Axis_Object.ConverterACSinglePhaseLossFault
   		elsif  	Axis_Object.ConverterACPhaseShortFault 			then temp_num:=S_CIPAxisFault.LEN+1; INSERT(Alarm_Texts[23],S_CIPAxisFault,temp_num,S_CIPAxisFault); // 	Axis_Object.ConverterACPhaseShortFault
   		elsif  	Axis_Object.ConverterPreChargeFault 			then temp_num:=S_CIPAxisFault.LEN+1; INSERT(Alarm_Texts[24],S_CIPAxisFault,temp_num,S_CIPAxisFault); // 	Axis_Object.ConverterPreChargeFault
   		elsif  	Axis_Object.BusRegulatorOvertemperatureFLFault 	then temp_num:=S_CIPAxisFault.LEN+1; INSERT(Alarm_Texts[25],S_CIPAxisFault,temp_num,S_CIPAxisFault); // 	Axis_Object.BusRegulatorOvertemperatureFLFault
   		elsif  	Axis_Object.BusRegulatorOvertemperatureULFault 	then temp_num:=S_CIPAxisFault.LEN+1; INSERT(Alarm_Texts[26],S_CIPAxisFault,temp_num,S_CIPAxisFault); // 	Axis_Object.BusRegulatorOvertemperatureULFault
   		elsif  	Axis_Object.BusRegulatorThermalOverloadFLFault 	then temp_num:=S_CIPAxisFault.LEN+1; INSERT(Alarm_Texts[27],S_CIPAxisFault,temp_num,S_CIPAxisFault); // 	Axis_Object.BusRegulatorThermalOverloadFLFault
   		elsif  	Axis_Object.BusRegulatorThermalOverloadULFault 	then temp_num:=S_CIPAxisFault.LEN+1; INSERT(Alarm_Texts[28],S_CIPAxisFault,temp_num,S_CIPAxisFault); // 	Axis_Object.BusRegulatorThermalOverloadULFault
   		elsif  	Axis_Object.BusRegulatorFault 					then temp_num:=S_CIPAxisFault.LEN+1; INSERT(Alarm_Texts[29],S_CIPAxisFault,temp_num,S_CIPAxisFault); // 	Axis_Object.BusRegulatorFault
   		elsif  	Axis_Object.BusModuleFault 						then temp_num:=S_CIPAxisFault.LEN+1; INSERT(Alarm_Texts[30],S_CIPAxisFault,temp_num,S_CIPAxisFault); // 	Axis_Object.BusModuleFault
   		elsif   Axis_Object.BusUndervoltageFLFault 				then temp_num:=S_CIPAxisFault.LEN+1; INSERT(Alarm_Texts[31],S_CIPAxisFault,temp_num,S_CIPAxisFault); // 	Axis_Object.BusUndervoltageFLFault
   		elsif  	Axis_Object.BusUndervoltageULFault 				then temp_num:=S_CIPAxisFault.LEN+1; INSERT(Alarm_Texts[32],S_CIPAxisFault,temp_num,S_CIPAxisFault); //  	Axis_Object.BusUndervoltageULFault
   		elsif  	Axis_Object.BusOvervoltageFLFault 				then temp_num:=S_CIPAxisFault.LEN+1; INSERT(Alarm_Texts[33],S_CIPAxisFault,temp_num,S_CIPAxisFault); // 	Axis_Object.BusOvervoltageFLFault
   		elsif  	Axis_Object.BusOvervoltageULFault 				then temp_num:=S_CIPAxisFault.LEN+1; INSERT(Alarm_Texts[34],S_CIPAxisFault,temp_num,S_CIPAxisFault); // 	Axis_Object.BusOvervoltageULFault
   		elsif  	Axis_Object.BusPowerLossFault 					then temp_num:=S_CIPAxisFault.LEN+1; INSERT(Alarm_Texts[35],S_CIPAxisFault,temp_num,S_CIPAxisFault); // 	Axis_Object.BusPowerLossFault
   		elsif  	Axis_Object.BusPowerBlownFuseFault 				then temp_num:=S_CIPAxisFault.LEN+1; INSERT(Alarm_Texts[36],S_CIPAxisFault,temp_num,S_CIPAxisFault); // 	Axis_Object.BusPowerBlownFuseFault
   		elsif  	Axis_Object.BusPowerLeakageFault 				then temp_num:=S_CIPAxisFault.LEN+1; INSERT(Alarm_Texts[37],S_CIPAxisFault,temp_num,S_CIPAxisFault); // 	Axis_Object.BusPowerLeakageFault
   		elsif  	Axis_Object.BusPowerSharingFault 				then temp_num:=S_CIPAxisFault.LEN+1; INSERT(Alarm_Texts[38],S_CIPAxisFault,temp_num,S_CIPAxisFault); // 	Axis_Object.BusPowerSharingFault
   		elsif  	Axis_Object.FeedbackSignalNoiseFLFault 			then temp_num:=S_CIPAxisFault.LEN+1; INSERT(Alarm_Texts[39],S_CIPAxisFault,temp_num,S_CIPAxisFault); // 	Axis_Object.FeedbackSignalNoiseFLFault
   		elsif  	Axis_Object.FeedbackSignalNoiseULFault 			then temp_num:=S_CIPAxisFault.LEN+1; INSERT(Alarm_Texts[40],S_CIPAxisFault,temp_num,S_CIPAxisFault); // 	Axis_Object.FeedbackSignalNoiseULFault
   		elsif  	Axis_Object.FeedbackSignalLossFLFault 			then temp_num:=S_CIPAxisFault.LEN+1; INSERT(Alarm_Texts[41],S_CIPAxisFault,temp_num,S_CIPAxisFault); // 	Axis_Object.FeedbackSignalLossFLFault
   		elsif  	Axis_Object.FeedbackSignalLossULFault 			then temp_num:=S_CIPAxisFault.LEN+1; INSERT(Alarm_Texts[42],S_CIPAxisFault,temp_num,S_CIPAxisFault); // 	Axis_Object.FeedbackSignalLossULFault
   		elsif  	Axis_Object.FeedbackDataLossFLFault 			then temp_num:=S_CIPAxisFault.LEN+1; INSERT(Alarm_Texts[43],S_CIPAxisFault,temp_num,S_CIPAxisFault); // 	Axis_Object.FeedbackDataLossFLFault
   		elsif  	Axis_Object.FeedbackDataLossULFault 			then temp_num:=S_CIPAxisFault.LEN+1; INSERT(Alarm_Texts[44],S_CIPAxisFault,temp_num,S_CIPAxisFault); // 	Axis_Object.FeedbackDataLossULFault
   		elsif  	Axis_Object.FeedbackDeviceFault 				then temp_num:=S_CIPAxisFault.LEN+1; INSERT(Alarm_Texts[45],S_CIPAxisFault,temp_num,S_CIPAxisFault); //  	Axis_Object.FeedbackDeviceFault
   		elsif  	Axis_Object.SensorFault 						then temp_num:=S_CIPAxisFault.LEN+1; INSERT(Alarm_Texts[46],S_CIPAxisFault,temp_num,S_CIPAxisFault); // 	Axis_Object.SensorFault
   		elsif  	Axis_Object.BrakeSlipFault 						then temp_num:=S_CIPAxisFault.LEN+1; INSERT(Alarm_Texts[47],S_CIPAxisFault,temp_num,S_CIPAxisFault); // 	Axis_Object.BrakeSlipFault
   		elsif  	Axis_Object.HardwareOvertravelPositiveFault 	then temp_num:=S_CIPAxisFault.LEN+1; INSERT(Alarm_Texts[48],S_CIPAxisFault,temp_num,S_CIPAxisFault); // 	Axis_Object.HardwareOvertravelPositiveFault
   		elsif   Axis_Object.HardwareOvertravelNegativeFault 	then temp_num:=S_CIPAxisFault.LEN+1; INSERT(Alarm_Texts[49],S_CIPAxisFault,temp_num,S_CIPAxisFault); // 	Axis_Object.HardwareOvertravelNegativeFault
   		elsif  	Axis_Object.ExcessivePositionErrorFault 		then temp_num:=S_CIPAxisFault.LEN+1; INSERT(Alarm_Texts[50],S_CIPAxisFault,temp_num,S_CIPAxisFault); // 	Axis_Object.ExcessivePositionErrorFault
   		elsif  	Axis_Object.ExcessiveVelocityErrorFault 		then temp_num:=S_CIPAxisFault.LEN+1; INSERT(Alarm_Texts[51],S_CIPAxisFault,temp_num,S_CIPAxisFault); // 	Axis_Object.ExcessiveVelocityErrorFault
   		elsif  	Axis_Object.OvertorqueLimitFault 				then temp_num:=S_CIPAxisFault.LEN+1; INSERT(Alarm_Texts[52],S_CIPAxisFault,temp_num,S_CIPAxisFault); // 	Axis_Object.OvertorqueLimitFault
   		elsif  	Axis_Object.UndertorqueLimitFault 				then temp_num:=S_CIPAxisFault.LEN+1; INSERT(Alarm_Texts[53],S_CIPAxisFault,temp_num,S_CIPAxisFault); // 	Axis_Object.UndertorqueLimitFault
   		elsif  	Axis_Object.ExcessiveBusVoltageErrorFault 		then temp_num:=S_CIPAxisFault.LEN+1; INSERT(Alarm_Texts[54],S_CIPAxisFault,temp_num,S_CIPAxisFault); // 	Axis_Object.ExcessiveBusVoltageErrorFault
   		elsif  	Axis_Object.AmbientTemperatureRiseFault 		then temp_num:=S_CIPAxisFault.LEN+1; INSERT(Alarm_Texts[55],S_CIPAxisFault,temp_num,S_CIPAxisFault); // 	Axis_Object.AmbientTemperatureRiseFault
   		elsif  	Axis_Object.IllegalControlModeFault 			then temp_num:=S_CIPAxisFault.LEN+1; INSERT(Alarm_Texts[56],S_CIPAxisFault,temp_num,S_CIPAxisFault); // 	Axis_Object.IllegalControlModeFault
   		elsif  	Axis_Object.EnableInputDeactivatedFault 		then temp_num:=S_CIPAxisFault.LEN+1; INSERT(Alarm_Texts[57],S_CIPAxisFault,temp_num,S_CIPAxisFault); // 	Axis_Object.EnableInputDeactivatedFault
   		elsif  	Axis_Object.ControllerInitiatedFault 			then temp_num:=S_CIPAxisFault.LEN+1; INSERT(Alarm_Texts[58],S_CIPAxisFault,temp_num,S_CIPAxisFault); // 	Axis_Object.ControllerInitiatedFault
   		elsif  	Axis_Object.ExternalInputFault 					then temp_num:=S_CIPAxisFault.LEN+1; INSERT(Alarm_Texts[59],S_CIPAxisFault,temp_num,S_CIPAxisFault); // 	Axis_Object.ExternalInputFault
   		elsif  	(Wrk_AxisState = 0 AND Sts_Faulted) 			then temp_num:=S_CIPAxisFault.LEN+1; INSERT(Alarm_Texts[60],S_CIPAxisFault,temp_num,S_CIPAxisFault); // 	Axis was not active while some fault occoured, therfor no error bits are set. why? only kinetix can explain..
   		elsif  	(Wrk_AxisState = 5 AND Sts_Faulted) 			then temp_num:=S_CIPAxisFault.LEN+1; INSERT(Alarm_Texts[61],S_CIPAxisFault,temp_num,S_CIPAxisFault); // 	Axis was not active while some fault occoured, therfor no error bits are set. why? only kinetix can explain..
   		elsif  	(Wrk_AxisState = 8 AND Sts_Faulted)				then temp_num:=S_CIPAxisFault.LEN+1; INSERT(Alarm_Texts[62],S_CIPAxisFault,temp_num,S_CIPAxisFault); // 	Axis was not active while some fault occoured, therfor no error bits are set. why? only kinetix can explain..
   		elsif  	Wrk_CIPAxisFault.63 							then temp_num:=S_CIPAxisFault.LEN+1; INSERT(Alarm_Texts[63],S_CIPAxisFault,temp_num,S_CIPAxisFault); // 	spare
   		end_if;
   	#endregion
   	/* Build begin of string */
   	temp_num:=Wrk_FaultMessage.LEN+1;
   	INSERT(S_FaultCode_Base,Wrk_FaultMessage,temp_num,Wrk_FaultMessage);
   	temp_num:=0;// set temp_num back to 0, since we dont need to keep track of this value.
   
   	/* S_ModuleFaultCode Contains data */
   	if S_ModuleFaultCode.LEN > 0 then
   		temp_num:=Wrk_FaultMessage.LEN+1;
   		INSERT(S_ModuleFaultCode,Wrk_FaultMessage,temp_num,Wrk_FaultMessage);
   		temp_num:=0;// set temp_num back to 0, since we dont need to keep track of this value.
   	end_if;
   	/* S_AxisFaultBits Contains data */
   	if S_AxisFaultBits.LEN > 0 then
   		temp_num:=S_AxisFaultBits.LEN+1;
   		INSERT(S_AxisFaultBits,Wrk_FaultMessage,temp_num,Wrk_FaultMessage);
   		temp_num:=0;// set temp_num back to 0, since we dont need to keep track of this value.
   	end_if;
   	/* S_MotionFaultBits Contains data */
   	if S_MotionFaultBits.LEN > 0 then
   		temp_num:=S_MotionFaultBits.LEN+1;
   		INSERT(S_MotionFaultBits,Wrk_FaultMessage,temp_num,Wrk_FaultMessage);
   		temp_num:=0;// set temp_num back to 0, since we dont need to keep track of this value.
   	end_if;
   	/* S_CIPAxisFault Contains data */
   	if S_CIPAxisFault.LEN > 0 then
   		temp_num:=S_CIPAxisFault.LEN+1;
   		INSERT(S_CIPAxisFault,Wrk_FaultMessage,temp_num,Wrk_FaultMessage);
   		temp_num:=0;// set temp_num back to 0, since we dont need to keep track of this value.
   	end_if;
   
   	if Wrk_FaultMessage <> Sts_FaultMessage then COP(Wrk_FaultMessage,Sts_FaultMessage,1); end_if;
   #endregion
   #region Controlled stop
   	if Inp_Stop AND SEQ_Stopping=0 then SEQ_Stopping:=10; end_if;
   	case SEQ_Stopping of
   		0: /* Waiting for command */
   			Sts_StandStill:=Axis_Object.VelocityStandstillStatus;
   		10: /* Check if axis is moving */
   			if 		Axis_Object.VelocityStandstillStatus then SEQ_Stopping:=0; end_if;// no motion, so therfor no stopping.
   			if NOT 	Axis_Object.VelocityStandstillStatus then SEQ_Stopping:=20; end_if;// Axis is moving
   		20: /* Save current position and Stop drive */
   			wrk_CurrentPosition:=0;																// clear previous stopping position.
   			wrk_CurrentPosition:=Axis_Object.ActualPosition;									// Save stopping position.
   			GSV(Axis,Axis_Object,MaximumDeceleration,wrk_Max_DecelRate);						// get max decel velocity²
   			if Cnf_DecelRate > wrk_Max_DecelRate then Cnf_DecelRate:=wrk_Max_DecelRate; end_if;	// if decel rate set by user is not within limits set highest limit.
   			if Cnf_DecelRate=0.0 then Cnf_DecelRate:=wrk_Max_DecelRate*0.01; end_if;				// if user forgot to set decel rate, set 1% of max decelrate.
   			if Cnf_DecelJerk=0.0 then Cnf_DecelJerk:=10; end_if;									// if user forgot to set Cnf_DecelJerk, set 10% of time.
   			MAS(
   				Axis_Object,
   				MAS_Axis,
   				All,
   				Yes,
   				Cnf_DecelRate,
   				Unitspersec2,
   				Yes,
   				Cnf_DecelJerk,
   				%ofTime
   			);
   			SEQ_Stopping:=25;
   		25: /* wait for feedback from MAS */
   			if MAS_Axis.EN AND MAS_Axis.PC then SEQ_Stopping:=30; end_if;
   			if MAS_Axis.EN AND MAS_Axis.ER then SEQ_Stopping:=999; end_if;
   		30: /* check if Cnf_RetrieveStoppingPositions is set */
   			Inp_Stop:=FALSE;		// feedback to user, execution was done.
   			if Cnf_RetrieveStoppingPositions then SEQ_Stopping:=40; else SEQ_Stopping:=0; end_if;
   		40: /* Move back to stoppping position */
   			GSV(Axis,Axis_Object,MaximumSpeed,wrk_MaximumSpeed);								// get max velocity
   			if Cnf_Retrieve_Speed=0 then Cnf_Retrieve_Speed:=wrk_MaximumSpeed*0.001; end_if;	// if user forgot to set speed, set 0.1% of max speed.
   			if Cnf_Retrieve_Accel=0 then Cnf_Retrieve_Accel:=wrk_Max_DecelRate*0.01; end_if;	// if user forgot to set accel rate, set 1% of max decelrate.
   			MAM(
   				Axis_Object,
   				MAM_Axis,
   				0/*absolute position*/,
   				wrk_CurrentPosition,
   				Cnf_Retrieve_Speed,
   				Unitspersec,
   				Cnf_Retrieve_Accel,
   				Unitspersec2,
   				Cnf_Retrieve_Accel,
   				Unitspersec2,
   				SCurve,
   				10,
   				10,
   				%ofTime,
   				0,
   				0,
   				0,
   				0,
   				0,
   				0
   			);
   			SEQ_Stopping:=45;
   		45: /* wait for feedback from MAM */
   			if MAM_Axis.EN AND MAM_Axis.PC then SEQ_Stopping:=0; end_if;
   			if MAM_Axis.EN AND MAM_Axis.ER then SEQ_Stopping:=999; end_if;
   		999: /* Error state */
   			Inp_Stop:=FALSE;		// feedback to user, execution was done.
   			if reset_ons.OutputBit then SEQ_Stopping:=0; end_if; // on reset set state back to 0.
   		else
   	end_case;
   #endregion
   
   
   
   
END_ROUTINE
END_ADD_ON_INSTRUCTION

ADD_ON_INSTRUCTION Substring   (* revision 1.0, vendor WPI *)
VAR_IN_OUT
   Input : STRING; {required}   // String to substring
END_VAR
VAR_INPUT
   From : INT; {required}   // where to start substringing
   End : DINT; {required}   // Where to end the substring
END_VAR
VAR_IN_OUT
   Result : STRING; {required}   // Result from substring
END_VAR
VAR
   i : DINT; {access None}   // local index
END_VAR

ROUTINE Logic   (* structured text *)
   #region Prevent controler fault
   		if From >= 80 	then From	:=80;	end_if;		// starting pos can never be higher then 80
   		if -1 	>= From then From	:=0; 	end_if;		// starting pos can never be lower then 0
   
   		if End >= 81 	then From	:=81;	end_if;		// ending pos can never be higher then 81
   		if -1 	>= End 	then End	:=1; 	end_if;		// ending pos can never be lower then 1
   	if From >= End then
   		End						:=	From+1;				// if end is lower or equal to from, no boundries are set for a substring. to prevent this add 1 to end to substring only 1 char.
   	end_if;
   #endregion
   #region Substring
   	#region clear previous data
   		for i := 0 to 81 do
   			Result.DATA[i] 		:=	0;					// set all data back to 0
   		end_for;
   		Result.LEN				:=	0;					// string length is set back to 0
   	#endregion
   	for i := From to End do
   		Result.DATA[i-From]		:=	Input.DATA[i];		// add substring data to Result, shift Index to start from Result.data[0] -> Result.data[1] -> Result.data[2] etc.
   	end_for;
   	Result.LEN					:=	End-From;			// set string length
   #endregion
END_ROUTINE
END_ADD_ON_INSTRUCTION

PROGRAM MainProgram   (* main routine MainRoutine *)

ROUTINE MainRoutine   (* ladder *)
END_ROUTINE
END_PROGRAM

PROGRAM SafetyProgram   (* main routine MainRoutine, safety *)

ROUTINE MainRoutine   (* ladder *)
END_ROUTINE
END_PROGRAM
